{attribute 'qualified_only'}
{attribute 'strict'}
TYPE BagMachineStatus:
(
    OFF := 0,
    BUSY := 1,
    READY := 2,
    BAG_READY := 3,
	MOVEIN_ENABLE	:= 4,
    BAG_INSERTED := 5,
	BAG_REMOVED := 6,
	GET_RESULT_FROM_CAMERA	:=7,
	RESET_CAMERA	:= 8,
	CAMERA_OK	:= 9,
	CAMERA_NG	:= 11,
    SUCCESS := 12,
    ERROR := 13,
	DONE	:=14
);
END_TYPE

(* stored: Version 1.1.0.1, ProductVersion 3.1.4024.12
   DUT BagMachineStatus: Id {cb7ae566-ce92-4914-a4d5-caf80dfbd1ff} *)
